// TwinCAT 3 PLC project PlcModel
// ProgramVersion: 3.1.4023.0
// libraries:
//   Tc2_Standard, * (Beckhoff Automation GmbH)
//   Tc2_System, * (Beckhoff Automation GmbH)
//   Tc3_Module, * (Beckhoff Automation GmbH)
// project tree:
//   GVLs/ ModelSetup.TcGVL
//   / PlcTask.TcTTO
//   POUs/ MAIN.TcPOU
// real-time tasks:
//   TASK PlcTask: cycle T#10ms, priority 20, ADS port 350
// I/O:
//   DEVICE Gerät 1 (EtherCAT Automation Protocol), AmsNetId 169.254.228.245.2.1
//     Box To Control (Publisher)
//     Box From Control (Subscriber)
// variable links:
//   Device 1 (EtherCAT Automation Protocol) <-> TcCOM Objects/Object1 (Vereinzelung)
//     Box From Control (Subscriber)/VereinzHub/Inputs/VarData[0,0] <-> Vereinzelung_U/Hw_ActUpOpen
//     Box From Control (Subscriber)/VereinzHub/Inputs/VarData[0,1] <-> Vereinzelung_U/Hw_ActUpClose
//     Box From Control (Subscriber)/VereinzHub/Inputs/VarData[1,0] <-> Vereinzelung_U/Hw_ActDownOpen
//     Box From Control (Subscriber)/VereinzHub/Inputs/VarData[1,1] <-> Vereinzelung_U/Hw_ActDownClose
//     Box To Control (Publisher)/VereinzSens/Outputs/VarData[0] <-> Vereinzelung_Y/Hw_SensorUp
//     Box To Control (Publisher)/VereinzSens/Outputs/VarData[1] <-> Vereinzelung_Y/Hw_SensorMiddle
//     Box To Control (Publisher)/VereinzSens/Outputs/VarData[2] <-> Vereinzelung_Y/Hw_SensorDown
//   Device 1 (EtherCAT Automation Protocol) <-> TcCOM Objects/Object2 (ModelConveyorWithLogic)
//     Box From Control (Subscriber)/BandHub/Inputs/VarData[0] <-> ModelConveyorWithLogic_U/HwStopper1
//     Box From Control (Subscriber)/BandHub/Inputs/VarData[1] <-> ModelConveyorWithLogic_U/HwStopper2
//     Box From Control (Subscriber)/BandHub/Inputs/VarData[2] <-> ModelConveyorWithLogic_U/HwStopper3
//     Box From Control (Subscriber)/DriveVelocity/Inputs/VarData[0] <-> ModelConveyorWithLogic_U/VelocityFromPLC
//     Box To Control (Publisher)/BandSens/Outputs/VarData[{0..3}] <-> ModelConveyorWithLogic_Y/HwSensor{1..4}  (4 links)
//     Box To Control (Publisher)/DriveCounterValue/Outputs/VarData[0] <-> ModelConveyorWithLogic_Y/CounterValueMotor
//     Box To Control (Publisher)/DriveState/Outputs/VarData[0] <-> ModelConveyorWithLogic_Y/DriveStateMotor
//   PlcModel/PlcModel Instance <-> TcCOM Objects/Object1 (Vereinzelung)
//     PlcTask Outputs/ModelSetup.samplingtime <-> Vereinzelung_U/SamplingTime
//     PlcTask Outputs/ModelSetup.signalCreateContainer <-> Vereinzelung_U/Signal_CreateContainer
//     PlcTask Outputs/ModelSetup.signalMaxPosAct <-> Vereinzelung_U/Signal_MaxPosAct
//     PlcTask Outputs/ModelSetup.signalMinPosAct <-> Vereinzelung_U/Signal_MinPosAct
//     PlcTask Outputs/ModelSetup.signalRevomeContainer <-> Vereinzelung_U/Signal_RemoveContainerOnConveyo
//   PlcModel/PlcModel Instance <-> TcCOM Objects/Object2 (ModelConveyorWithLogic)
//     PlcTask Outputs/ModelSetup.samplingtime <-> ModelConveyorWithLogic_U/SamplingTime
//     PlcTask Outputs/ModelSetup.signalCreateContainerConveyor <-> ModelConveyorWithLogic_U/SignalCreateContainer
//     PlcTask Outputs/ModelSetup.signalRevomeContainerConveyor <-> ModelConveyorWithLogic_U/SignalRemoveContainer

CONFIGURATION PlcModel
    RESOURCE PLC ON TwinCAT3
        TASK PlcTask(INTERVAL := T#10ms, PRIORITY := 20);
        PROGRAM MAIN WITH PlcTask : MAIN;
    END_RESOURCE
END_CONFIGURATION

// ---- GVLs/ModelSetup.TcGVL
{attribute 'qualified_only'}
VAR_GLOBAL
	samplingtime 			AT%Q* : LREAL := 0.01;
	
	signalCreateContainer 	AT%Q* : BOOL;
	signalRevomeContainer 	AT%Q* : BOOL;
	signalMinPosAct 		AT%Q* : LREAL := 0;
	signalMaxPosAct 		AT%Q* : LREAL := 10;
	
	// Conveyor
	signalCreateContainerConveyor 	AT%Q* : BOOL;
	signalRevomeContainerConveyor 	AT%Q* : BOOL;
	
	velo AT%Q* : INT;
END_VAR

// ---- POUs/MAIN.TcPOU
PROGRAM MAIN
VAR
	counter : INT;
END_VAR

counter := counter +1;

END_PROGRAM
